INTERFACE I_XP_System_PLC EXTENDS I_CH_Object

METHOD CheckTargetExists : BOOL //Return TRUE if target is existing
VAR_INPUT
	sStation	: STRING; //Group of the targed station or LUID
END_VAR
END_METHOD

METHOD Disable : I_CH_Feedback
VAR_INPUT
END_VAR
END_METHOD

{attribute 'monitoring':='call'}
PROPERTY Disabled : BOOL
GET
END_GET
END_PROPERTY

METHOD Enable : I_CH_Feedback
VAR_INPUT
END_VAR
END_METHOD

{attribute 'monitoring':='call'}
PROPERTY Enabled : BOOL
GET
END_GET
END_PROPERTY

{attribute 'monitoring':='call'}
PROPERTY Enviroment : I_XP_Environment
GET
END_GET
END_PROPERTY

{attribute 'monitoring':='call'}
PROPERTY Feedback : CHALET_BaseComponents.I_CH_Feedback
GET
END_GET
END_PROPERTY

METHOD Initialize : HRESULT
VAR_INPUT
END_VAR
END_METHOD

{attribute 'monitoring':='call'}
PROPERTY Initialized : BOOL
GET
END_GET
END_PROPERTY

{attribute 'monitoring':='call'}
PROPERTY Movers : CHALET_BaseComponents.I_CH_LIST
GET
END_GET
END_PROPERTY

METHOD Station : I_XP_Station_PLC
VAR_INPUT
	sLUID : STRING;
END_VAR
END_METHOD

{attribute 'monitoring':='call'}
PROPERTY Stations : CHALET_BaseComponents.I_CH_LIST
GET
END_GET
END_PROPERTY

{attribute 'monitoring':='call'}
PROPERTY Tracks : CHALET_BaseComponents.I_CH_LIST
GET
END_GET
END_PROPERTY

{attribute 'monitoring':='call'}
PROPERTY Triggers : CHALET_BaseComponents.I_CH_LIST
GET
END_GET
END_PROPERTY

METHOD Update : HRESULT
VAR_INPUT
END_VAR
END_METHOD

//Return TRUE if unique station id is valid. if false, interfacepointer is zero -> fatal error
METHOD ValidLUID : BOOL
VAR_INPUT
	sLUID : STRING;
END_VAR
END_METHOD

{attribute 'monitoring':='call'}
PROPERTY Zones : CHALET_BaseComponents.I_CH_LIST
GET
END_GET
END_PROPERTY

END_INTERFACE

(* stored: Version 1.1.0.1, ProductVersion 3.1.4024.12
   Itf I_XP_System_PLC: Id {c3b3d3ce-c3c0-4441-bc62-ab81925683e6}
   Method CheckTargetExists: Id {41af54e4-98a3-42b3-a270-0f5a5953c6eb}
   Method Disable: Id {0e1c17f7-3e58-40a2-9be7-754489d0378a}
   Property Disabled: Id {f3895e35-e9a7-4cf9-a54f-bdfaf156d398}
   Get Get: Id {1069656a-54de-4969-868d-b4d23d51a907}
   Method Enable: Id {b7d5fbd1-5b07-42a2-8c1a-086f194cd652}
   Property Enabled: Id {b42af01e-628a-4469-86e2-a89c4d5bb60f}
   Get Get: Id {a16c6594-ee7f-4500-a7d6-fb38a5441e50}
   Property Enviroment: Id {3af0d81b-396b-4659-8386-10bee2c5c9c2}
   Get Get: Id {e36241ae-c759-4204-9626-3a54ce86185c}
   Property Feedback: Id {170543fd-4784-4c2f-86da-1f2e4449e206}
   Get Get: Id {257eba3d-00ce-4a79-9f6a-e3956376d85e}
   Method Initialize: Id {b2268470-01d2-4e0d-a4ab-dae39eacd787}
   Property Initialized: Id {fdcd6d33-ed24-4025-8271-1ee3999b78ed}
   Get Get: Id {d5c068fc-3605-452e-be7e-2a99229d27fd}
   Property Movers: Id {eb1e997d-a42b-4926-a204-df00717ba322}
   Get Get: Id {e2e7ae6b-0a08-4719-9298-403b515ebd6f}
   Method Station: Id {4ab23b5f-6de5-43ad-bb89-4891f9681ff6}
   Property Stations: Id {72cbf4b8-aca0-4ec3-b014-b877cfe731c1}
   Get Get: Id {b0e6f6ff-8d89-4f2b-8235-1909b8f695e9}
   Property Tracks: Id {7afd3d84-45ba-4e25-ac84-29da3d991836}
   Get Get: Id {d36e3d85-61b4-4b63-a0d0-33b491fca692}
   Property Triggers: Id {413ec768-c88f-47f1-a0e8-c8b78e083282}
   Get Get: Id {45bd0021-e4b3-4d24-93dc-cf4065d4dad1}
   Method Update: Id {09407e8b-d7ce-4a68-a4f9-b085d0bf0c23}
   Method ValidLUID: Id {175dfe5d-22be-4bfd-961a-4b5a744f93c8}
   Property Zones: Id {a7842daf-3b5c-4056-b978-11416a243f2c}
   Get Get: Id {13bae06b-dfd1-442c-8d06-8e18d8364428} *)
